(* PLC project Sin nombre, Desconocido Sin nombre 1 *)
(* stored: creationDateTime 2020-07-07T11:10:56, modificationDateTime 2020-07-07T11:53:19 *)

PROGRAM io_esp_01
  VAR
    IN AT %IX100.0 : BOOL;
    OUT AT %QX100.3 : BOOL;
  END_VAR

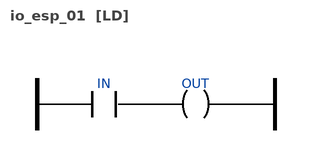
(* LD diagram, written out as Structured Text *)
OUT := IN;
END_PROGRAM

CONFIGURATION Config0
  RESOURCE Res0 ON PLC
    TASK task0(INTERVAL := T#20ms, PRIORITY := 0);
    PROGRAM instance0 WITH task0 : io_esp_01;
  END_RESOURCE
END_CONFIGURATION
